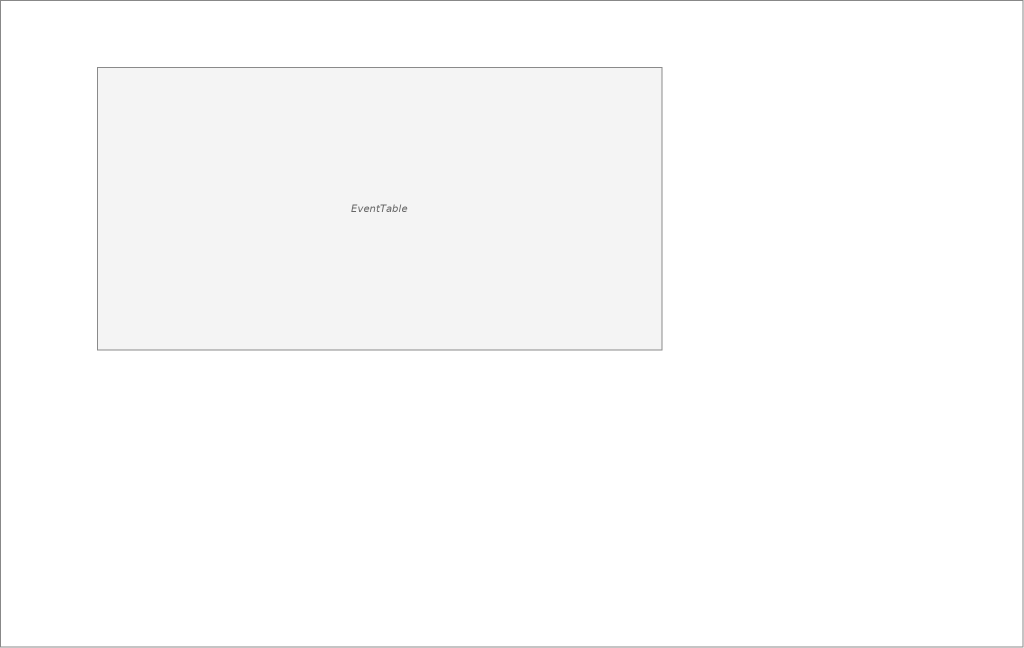
VISUALIZATION Alarmy  // 1024x648
    EventTable (97,67 565x283)
        p1690906150: Class
        p3258520714: Date
        p2231227367: Time
        p3993844394: Message
        p2076579579: Details
        p3558512729: aEventsSimple
        p3921149237: m_pDataArray..pArray
END_VISUALIZATION

(* stored: Version 1.1.0.1, ProductVersion 3.1.4022.12
   Visu Alarmy: Id {9162b894-3287-481f-b226-7b9de68c6c01} *)
